FUNCTION_BLOCK FB_SaMElementStopping EXTENDS FB_SaMElement
VAR
END_VAR

METHOD FB_init : BOOL
VAR_INPUT
	bInitRetains : BOOL; // if TRUE, the retain variables are initialized (warm start / cold start)
	bInCopyCode : BOOL;  // if TRUE, the instance afterwards gets moved into the copy code (online change)
END_VAR
THIS^.SetText (eLocation := E_BaseLocation.pl, wsDescription := "Zatrzymywanie");
THIS^.SetText (eLocation := E_BaseLocation.en, wsDescription := "Stopping");
THIS^.SetText (eLocation := E_BaseLocation.de, wsDescription := "Anhalten");
THIS^.SetName (stName := THIS^.GetTexts ());
END_METHOD

METHOD PUBLIC InvokeStateForTopElement : BOOL
VAR_INPUT
	itfTopElement		: ITF_BaseSaMStateMethod;
END_VAR
InvokeStateForTopElement	:= itfTopElement.SP_Stopping ();
END_METHOD

END_FUNCTION_BLOCK

(* stored: Version 1.1.0.1
   POU FB_SaMElementStopping: Id {a338b75d-6bec-0e21-0e98-ef0d6f0bcdbc}, SpecialFunc None
   Method FB_init: Id {1b1c099c-8d81-0204-2048-91a85295021d}
   Method InvokeStateForTopElement: Id {a716ed17-84a0-0b94-3043-9c9655754cc2} *)
